FUNCTION Tanque : bool
VAR_INPUT
END_VAR
VAR
END_VAR

//Si tengo piez delante
// bajo nivel de tanque (apertura de valvula) durante X segundos
// Paro y devuelvo true (listo para continuar)

(*COMPROBACIONES 
 	* Que haya siempre fluido en el tanque
	* Tener pieza delante
*)

END_FUNCTION

(* stored: Version 1.1.0.1, ProductVersion 3.1.4024.15
   POU Tanque: Id {275e80ce-beff-4c0a-aa36-8b287ee0e914}, SpecialFunc None *)
